FUNCTION xdotc_iq : LREAL
VAR_INPUT
    b_n: DINT;
    x: ARRAY [0..35] OF LREAL;
    ix0: DINT;
    y: ARRAY [0..35] OF LREAL;
    iy0: DINT;
END_VAR
VAR
    ix: DINT;
    iy: DINT;
    k: DINT;
END_VAR

xdotc_iq := 0.0;
IF b_n >= 1 THEN 
    ix := ix0;
    iy := iy0;
    k := 0;
    WHILE k <= (b_n - 1) DO
        xdotc_iq := (x[ix - 1] * y[iy - 1]) + xdotc_iq;
        ix := ix + 1;
        iy := iy + 1;
        k := k + 1;
    END_WHILE;
END_IF;

END_FUNCTION

(* stored: Version 1.1.0.1, ProductVersion 3.1.4024.12
   POU xdotc_iq: Id {0c7bc3ca-91cf-4047-afd3-251b6bbdbd67}, SpecialFunc None *)
